{attribute addProperty BoxType "EL5101--0000"}
{attribute addProperty Id "CtrlAT %Q*USINT811ValueAT %Q*UINT1622"}
{attribute addProperty CRC "1296992566"}
{attribute addProperty SizeInBites "24"}
{attribute addProperty SizeInBytes "3"}
TYPE Channel_4D4E8936 :
STRUCT
	{attribute addProperty Name "Ctrl"}
	Ctrl AT %Q* : USINT;
	{attribute addProperty Name "Value"}
	Value AT %Q* : UINT;
END_STRUCT
END_TYPE

(* stored: Version 1.2.0.0, ProductVersion 3.1.4024.9
   DUT Channel_4D4E8936: Id {241cd80b-6afa-4c5e-931c-5ff79b0c24a1} *)
